(* PLC project CoDeSys Ver 3.x Dbm Translations, Hydac System GmbH PdtCodeBuilder.dll 1.2.7.80 *)
(* stored: companyURL http://www.hydac.com/, contentDescription This content was automatically generated. Please do not edit., creationDateTime 2025-04-18T16:40:50.760 *)

